INTERFACE I_Concater

METHOD PUBLIC Clear : I_Concater
END_METHOD

METHOD PUBLIC GetString : STRING
END_METHOD

METHOD PUBLIC L : I_Concater
VAR_INPUT
    part : STRING;
END_VAR
END_METHOD

METHOD PUBLIC V : I_Concater
VAR_INPUT
    part : ANY;
END_VAR
END_METHOD

END_INTERFACE

(* stored: Version 1.1.0.1, ProductVersion 3.1.4024.12
   Itf I_Concater: Id {9ca42f3e-4c63-43e8-b01f-4d34b6fee744}
   Method Clear: Id {df0f2655-eaad-40bc-bc5c-606fedcf3e5b}
   Method GetString: Id {1989d606-e0f7-4373-b246-6aa0f6608f16}
   Method L: Id {68af6fe8-6055-493a-8622-a72f6266ea28}
   Method V: Id {c45fffae-2b88-4048-a002-c50ad539606c} *)
